(*

.. <legal notes>

legal notes
=================
| SPDX-FileCopyrightText: © 2025 Oleksandr Tiutyk <trofimich@gmail.com>
| SPDX-License-Identifier: LGPL-3.0-only
| For details check: LGPL-3.0-only_

.. _LGPL-3.0-only: https://www.gnu.org/licenses/lgpl-3.0.en.html

.. </legal notes>

*)

{attribute 'no_explicit_call' := 'do not call this function block directly'} 
FUNCTION_BLOCK ABSTRACT AbortableTask EXTENDS Object IMPLEMENTS IAbortableTask
VAR
	_StateChanged : BOOL;

	_Running : BOOL;

	_Done : BOOL;
	
	_Aborting : BOOL;	
	_Aborted : BOOL;
	_AbortReason : ERROR_MESSAGE;
	
	_Error : BOOL;	
	_ErrorMessage : ERROR_MESSAGE;	
END_VAR

{attribute 'monitoring' := 'call'}
{attribute 'OPC.UA.DA.Property' := '1'}
{attribute 'OPC.UA.DA.Access' := '1'}
PROPERTY FINAL Aborted : BOOL
GET
Aborted := _Aborted;
END_GET
END_PROPERTY

{attribute 'monitoring' := 'call'}
{attribute 'OPC.UA.DA.Property' := '1'}
{attribute 'OPC.UA.DA.Access' := '1'}
PROPERTY FINAL Aborting : BOOL
GET
Aborting := _Aborting;
END_GET
END_PROPERTY

{attribute 'monitoring' := 'call'}
{attribute 'OPC.UA.DA.Property' := '1'}
{attribute 'OPC.UA.DA.Access' := '1'}
PROPERTY FINAL AbortReason : REFERENCE TO ERROR_MESSAGE
GET
AbortReason REF= _AbortReason;
END_GET
END_PROPERTY

{attribute 'monitoring' := 'call'}
{attribute 'OPC.UA.DA.Property' := '1'}
{attribute 'OPC.UA.DA.Access' := '1'}
PROPERTY FINAL Busy : BOOL
GET
Busy := _Running OR_ELSE _Aborting;
END_GET
END_PROPERTY

{attribute 'monitoring' := 'call'}
{attribute 'OPC.UA.DA.Property' := '1'}
{attribute 'OPC.UA.DA.Access' := '1'}
PROPERTY FINAL Done : BOOL
GET
Done := _Done;
END_GET
END_PROPERTY

{attribute 'monitoring' := 'call'}
{attribute 'OPC.UA.DA.Property' := '1'}
{attribute 'OPC.UA.DA.Access' := '1'}
PROPERTY FINAL Error : BOOL
GET
Error := _Error;
END_GET
END_PROPERTY

{attribute 'monitoring' := 'call'}
{attribute 'OPC.UA.DA.Property' := '1'}
{attribute 'OPC.UA.DA.Access' := '1'}
PROPERTY FINAL ErrorMessage : REFERENCE TO ERROR_MESSAGE
GET
ErrorMessage REF= _ErrorMessage;
END_GET
END_PROPERTY

METHOD FINAL Execute 
VAR
	done : BOOL;
	
	exceptionCode : __SYSTEM.ExceptionCode;
	
	exception : IException;	
	
	errorMessage : ERROR_MESSAGE;
END_VAR
_StateChanged := FALSE;

__TRY
	IF Busy THEN
		IF _Running THEN
			OnRunning(FALSE, done => done);
			
			IF done THEN
				setDoneState();
			END_IF		
		ELSE
			OnAborting(FALSE, done => done);
			
			IF done THEN
				setAbortedState();
			END_IF		
		END_IF
	END_IF
__CATCH(exceptionCode)
	handleException(exceptionCode);
__ENDTRY
END_METHOD

METHOD PRIVATE handleException
VAR_INPUT
	exceptionCode : __SYSTEM.ExceptionCode;
END_VAR
VAR
	exception : IException;
END_VAR
exception := ExceptionManager.GetLastException(exceptionCode);

__TRY
	OnError();
__CATCH
__ENDTRY

_ErrorMessage := exception.GetMessage();
	
IF NOT _Error THEN
	LogManager.TryLogMessage(WideStringHelper.ConcatStrings255("Task '", Name, "' failed at ", TO_WSTRING(SystemDateTimeManager.SystemLocalDateTime)), LOG_CATEGORY.SUCCESS, TO_WSTRING(ClassName), "Task", "TaskFailed");
	
	_StateChanged := TRUE;
END_IF

_Running := FALSE;

_Done := FALSE;

_Aborting := FALSE;	
_Aborted := FALSE;
_AbortReason := "";

_Error := TRUE;		

ExceptionManager.Throw(exception);
END_METHOD

{attribute 'monitoring' := 'call'}
{attribute 'OPC.UA.DA.Property' := '1'}
{attribute 'OPC.UA.DA.Access' := '1'}
PROPERTY ABSTRACT Name : WSTRING
GET
END_GET
END_PROPERTY

METHOD PROTECTED ABSTRACT OnAborting 
VAR_INPUT
	isStart : BOOL;
END_VAR
VAR_OUTPUT
	done : BOOL;
END_VAR
END_METHOD

METHOD PROTECTED OnError
END_METHOD

METHOD PROTECTED ABSTRACT OnRunning 
VAR_INPUT
	isStart : BOOL;
END_VAR
VAR_OUTPUT
	done : BOOL;
END_VAR
END_METHOD

{attribute 'monitoring' := 'call'}
{attribute 'OPC.UA.DA.Property' := '1'}
{attribute 'OPC.UA.DA.Access' := '1'}
PROPERTY FINAL Running : BOOL
GET
Running := _Running;
END_GET
END_PROPERTY

METHOD PRIVATE FINAL setAbortedState
IF NOT _Aborted THEN
	LogManager.TryLogMessage(WideStringHelper.ConcatStrings255("Task '", Name, "' aborted at ", TO_WSTRING(SystemDateTimeManager.SystemLocalDateTime)), LOG_CATEGORY.SUCCESS, TO_WSTRING(ClassName), "Task", "TaskAborted");

	_StateChanged := TRUE;
END_IF

_Running := FALSE;

_Done := FALSE;

_Aborting := FALSE;	
_Aborted := TRUE;

_Error := FALSE;	
_ErrorMessage := "";
END_METHOD

METHOD PRIVATE FINAL setAbortingState
VAR_IN_OUT CONSTANT 
	reason : ERROR_MESSAGE;
END_VAR
IF NOT _Aborting THEN
	LogManager.TryLogMessage(WideStringHelper.ConcatStrings255("Task '", Name, "' abort started at ", TO_WSTRING(SystemDateTimeManager.SystemLocalDateTime)), LOG_CATEGORY.SUCCESS, TO_WSTRING(ClassName), "Task", "TaskAbortStarted");

	_StateChanged := TRUE;
END_IF

_Running := FALSE;

_Done := FALSE;

_Aborting := TRUE;	
_Aborted := FALSE;
_AbortReason := reason;

_Error := FALSE;	
_ErrorMessage := "";
END_METHOD

METHOD PRIVATE FINAL setDoneState
IF NOT _Done THEN
	LogManager.TryLogMessage(WideStringHelper.ConcatStrings255("Task '", Name, "' done at ", TO_WSTRING(SystemDateTimeManager.SystemLocalDateTime)), LOG_CATEGORY.SUCCESS, TO_WSTRING(ClassName), "Task", "TaskDone");
	
	_StateChanged := TRUE;
END_IF

_Running := FALSE;

_Done := TRUE;

_Aborting := FALSE;	
_Aborted := FALSE;
_AbortReason := "";

_Error := FALSE;	
_ErrorMessage := "";
END_METHOD

METHOD PRIVATE FINAL setRunningState
IF NOT _Running THEN
	LogManager.TryLogMessage(WideStringHelper.ConcatStrings255("Task '", Name, "' started at ", TO_WSTRING(SystemDateTimeManager.SystemLocalDateTime)), LOG_CATEGORY.SUCCESS, TO_WSTRING(ClassName), "Task", "TaskStarted");
	
	_StateChanged := TRUE;
END_IF

_Running := TRUE;

_Done := FALSE;

_Aborting := FALSE;	
_Aborted := FALSE;
_AbortReason := "";

_Error := FALSE;	
_ErrorMessage := "";
END_METHOD

METHOD FINAL Start
VAR
	done : BOOL;

	exceptionCode : __SYSTEM.ExceptionCode;
	
	exception : IException;

	errorMessage : ERROR_MESSAGE;	
END_VAR
__TRY
	setRunningState();
	
	OnRunning(TRUE, done => done);

	IF done THEN
		setDoneState();
	END_IF
__CATCH(exceptionCode)
	handleException(exceptionCode);
__ENDTRY
END_METHOD

METHOD FINAL StartAbort
VAR_INPUT 
	reason : ERROR_MESSAGE := "";
END_VAR
VAR
	done : BOOL;

	exceptionCode : __SYSTEM.ExceptionCode;
	
	exception : IException;

	errorMessage : ERROR_MESSAGE;	
END_VAR
IF NOT Running THEN
	RETURN;
END_IF

__TRY
	setAbortingState(reason);
	
	OnAborting(TRUE, done => done);

	IF done THEN
		setAbortedState();
	END_IF
__CATCH(exceptionCode)
	handleException(exceptionCode);
__ENDTRY
END_METHOD

{attribute 'monitoring' := 'call'}
{attribute 'OPC.UA.DA.Property' := '1'}
{attribute 'OPC.UA.DA.Access' := '1'}
PROPERTY FINAL StateChanged : BOOL
GET
StateChanged := _StateChanged;
END_GET
END_PROPERTY

END_FUNCTION_BLOCK

(* stored: Version 1.1.0.1
   POU AbortableTask: Id {3fcb82bf-fcc2-4c60-ab58-32776172ce5b}, SpecialFunc None
   Folder Members to override: Id {76112447-5878-4246-92fb-0910ffa3ef2d}
   Folder Service members: Id {6b1a5589-8d7c-4542-877b-5fcd2d9b2fbd}
   Property Aborted: Id {205fba08-26d2-4312-a96e-e17dee6c923f}
   Get Get: Id {9f8851fa-4d24-41c2-b7cf-fd9ecc9bdb84}
   Property Aborting: Id {c0530bff-30c3-4c28-990a-6e7a951c38e9}
   Get Get: Id {c76d8074-3a6c-4ceb-839f-e729688d48e1}
   Property AbortReason: Id {62b5d978-3b39-4864-a514-bb07423cf0e2}
   Get Get: Id {e89b4f7e-5119-407b-92c1-18a61068d8bb}
   Property Busy: Id {e3f55a84-6dc8-42a8-870b-cbc03d5ce896}
   Get Get: Id {9b0f9833-3b49-48b8-9041-0090b996669f}
   Property Done: Id {b95d743b-c72e-4bcb-a404-c7e3e4a6a37e}
   Get Get: Id {bfaa887d-c314-4518-a171-41d0308d56ff}
   Property Error: Id {3d54590f-9d24-46b4-9724-32260ce4207a}
   Get Get: Id {998b8321-1744-4a0a-b9cf-78a20c7dc6e5}
   Property ErrorMessage: Id {e92b95ec-4a2f-46a9-85eb-1f48df75a257}
   Get Get: Id {82e42fe0-1017-4cc0-a630-23020b73322e}
   Method Execute: Id {356dfaf1-5836-4634-88c3-9adf266fe2b8}
   Method handleException: Id {87f22517-b446-496a-a773-92d534ab21f6}
   Property Name: Id {6fc84b72-bae7-48c4-9b6d-21dd2d8602d7}
   Get Get: Id {159969ce-3ca4-45c0-a82e-3687a3ad2fff}
   Method OnAborting: Id {bd8eb179-c550-42d5-a679-2b68c1503c0e}
   Method OnError: Id {c12cd4b4-6b5e-40a4-9547-4538d1fad656}
   Method OnRunning: Id {a15599f5-e9ad-4bc1-b827-e975fc966d86}
   Property Running: Id {dda6cb05-0e58-4715-8fa9-9ed4428ca958}
   Get Get: Id {ac4bced3-fa18-48d8-a5d4-4beba0226ec1}
   Method setAbortedState: Id {fac00809-31d6-4f90-8e02-b442214ce266}
   Method setAbortingState: Id {dc660dfe-c65d-4d91-bb97-ccc531a7b715}
   Method setDoneState: Id {5a91bd28-905f-4ff0-ac15-4afd240589a6}
   Method setRunningState: Id {8ba032d1-b467-4f29-94d8-e5d440995321}
   Method Start: Id {5e4f958e-3441-449c-a3ee-2bfa2bc2b0b1}
   Method StartAbort: Id {f4d5eddb-0774-4410-8518-af02c1510410}
   Property StateChanged: Id {5df375fb-8678-4172-86a8-056cc8dfa2cd}
   Get Get: Id {68fadd26-a99e-461e-8aa1-2b482d0dd654} *)
